// Mitsubishi GX Works2 project: RS232_Non_Protocol   PLC: Q06UDV
// RS232_Non_Protocol

PROGRAM MAIN
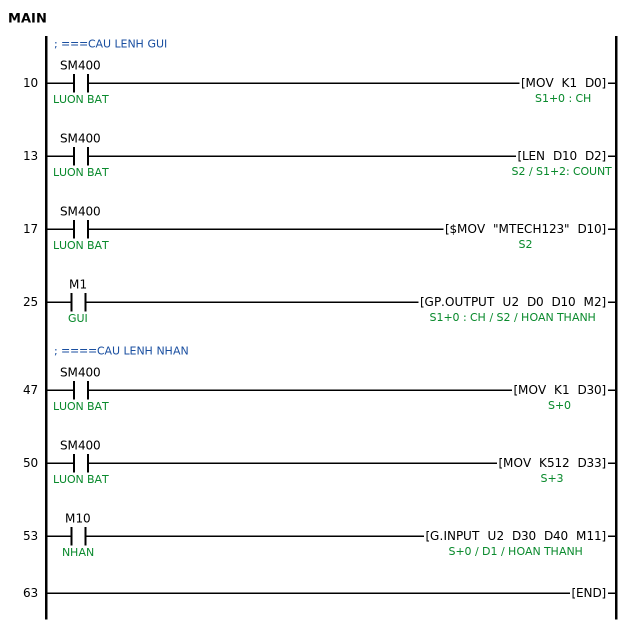
; ===CAU LENH GUI
10    LD      SM400  ; LUON BAT
      MOV     K1 D0  ; S1+0 : CH
13    LD      SM400  ; LUON BAT
      LEN     D10 D2  ; S2 / S1+2: COUNT
17    LD      SM400  ; LUON BAT
      $MOV    "MTECH123" D10
25    LD      M1  ; GUI
      GP.OUTPUT U2 D0 D10 M2  ; HOAN THANH
; ====CAU LENH NHAN
47    LD      SM400  ; LUON BAT
      MOV     K1 D30  ; S+0
50    LD      SM400  ; LUON BAT
      MOV     K512 D33  ; S+3
53    LD      M10  ; NHAN
      G.INPUT U2 D30 D40 M11  ; D1 / HOAN THANH
63    END
END_PROGRAM
